VAR_GLOBAL
// Inputs:

Queue	: DUT_RECIPEORDER;

//Outputs:

Offer	: ARRAY [0..OfferCnt] OF DUT_RECIPEOFFER;

// ProductionList

Task	: ARRAY [0..TaskCnt] OF DUT_TASK;
END_VAR

(* stored: Version 1.1.0.1, ProductVersion 3.1.0.25
   GVL I_O_GVL: Id {4dfb039f-3452-4ac3-9be1-1665c3d246ae} *)
